Fanuc KAREL source: t_arrfunc2.kl

PROGRAM TARRFUNC2
%NOLOCKGROUP
VAR
 gb: ARRAY[6] OF BOOLEAN
ROUTINE fbool(a: BOOLEAN): ARRAY[6] OF BOOLEAN
VAR
 t: ARRAY[6] OF BOOLEAN
BEGIN
 t[1] = a
 RETURN(t)
END fbool
BEGIN
 gb = fbool(TRUE)
END TARRFUNC2
